FUNCTION F_StopAnalogRamping_ForRecipe
VAR
	i: INT;
END_VAR

FOR i:= 1 TO E_aAnalogInputIO_Index.E_PV_EPC_04 DO
	IF 0.0 < GVL_IO.aAnalogController[i].maxValue THEN
		GVL_IO.aAnalogController[i].cvController.input.restart := TRUE;
		GVL_IO.aAnalogController[i].cvController.input.rampTime := 1; 
		GVL_IO.aAnalogController[i].cvController.input.targetValue := GVL_IO.aAnalogController[i].cv;
	END_IF
END_FOR

FOR i:= E_aAnalogInputIO_Index.E_PV_Susceptor_Temp TO E_aAnalogInputIO_Index.E_PV_susceptorRotation DO
	GVL_IO.aAnalogController[i].cvController.input.restart := TRUE;
	GVL_IO.aAnalogController[i].cvController.input.rampTime := 1;
	GVL_IO.aAnalogController[i].cvController.input.targetValue := GVL_IO.aAnalogController[i].cv;
END_FOR

END_FUNCTION

(* stored: Version 1.1.0.1, ProductVersion 3.1.4026.11
   POU F_StopAnalogRamping_ForRecipe: Id {894f4883-78ef-41b6-90b5-91f6e5cdbce2}, SpecialFunc None *)
